{region '#Template'}
	{attribute 'Version' := '6.0.0.0'}
	{attribute 'Tags' := '"LCID": "1031", "Text": "AC, Plant, AHU, Lüftungsanlage"'}
	{attribute 'Tags' := '"LCID": "1033", "Text": "AC, Plant, AHU, Air handling unit"'}
	{attribute 'Using' := '"Type": "Template", "URI": "Priority"'}		 
	{attribute 'Using' := '"Type": "Template", "URI": "Site"'}
	{attribute 'Using' := '"Type": "Template", "URI": "E_BA_AC_OpMod01"'}
	{attribute 'Using' := '"Type": "Template", "URI": "E_BA_AC_PlantStep01"'}
	{attribute 'Description' := '"LCID": "1031", "Text": "Ventilator druckgesteuert, Einfache Abluft/Zuluftkaskade, Vorerhitzer, ERC Platte, Kühler "'}
	{attribute 'Description' := '"LCID": "1033", "Text": "Fan pressure controlled, Simple extract air/supply air cascade, PreHeater, ERC Plate, Cooler"'}
{endregion}
FUNCTION_BLOCK FB_BA_AHU_1st_10 EXTENDS FB_BA_View
VAR_INPUT CONSTANT	
	TOuA					: FB_BA_SensorAnalog;			
	TExhA					: FB_BA_SensorAnalog;	
	TSuA					: FB_BA_SensorAnalog;	
	TExtA					: FB_BA_SensorAnalog;								
	TRm						: FB_BA_SensorAnalog;	

	DiffPrssOuAFilt			: FB_BA_SensorAnalog;											
	FiltOuAMonit			: FB_BA_Hys_21;							
	DiffPrssExtAFilt		: FB_BA_SensorAnalog;				
	FiltExtAMonit			: FB_BA_Hys_21;	

	OuADmp					: FB_BA_AC_Dmp2P;	
	SuAPrss					: FB_BA_SensorAnalog;	
	SuADiffPrss				: FB_BA_SensorAnalog;		
	SuAFan					: FB_BA_AC_FanCtl;	
	SuADiffPrssMonit		: FB_BA_FdbAnalog;								

	ExhADmp					: FB_BA_AC_Dmp2P;	
	ExtAPrss				: FB_BA_SensorAnalog;	
	ExtADiffPrss			: FB_BA_SensorAnalog;		
	ExtAFan					: FB_BA_AC_FanCtl;								
	ExtADiffPrssMonit		: FB_BA_FdbAnalog;

	PreHtr					: FB_BA_AC_PreHtr;	
	Erc						: FB_BA_AC_ErcPl_02;								
	Col						: FB_BA_AC_ColT_02;								

	SpTRm					: FB_BA_Scale_04_Y2_3;	
	TCasCtrl				: FB_BA_AC_TCasCtrl_01;										 								

	SumNgtCol				: FB_BA_AC_SumNgtCol;	
	OpMod					: FB_BA_AC_OpMod1St;	

	PlantLock				: FB_BA_PlantLock;	

	PlantCmd				: FB_BA_AC_PlantCmd_AHU_1st_10;	

	TSeqLink				: FB_BA_AC_SeqT;
	stTSeqLink				: ST_BA_SeqLink;	//	Sequenz Link Struktur	//	Sequence link structure		
	
	arrAggregate			: ARRAY [1..MAX(1,BA_Param.nMaxAggregate)] OF ST_BA_Aggregate;

END_VAR
VAR // added by the converter: edge detectors and wires of the graphical bodies
    _w1 : ANY;
END_VAR

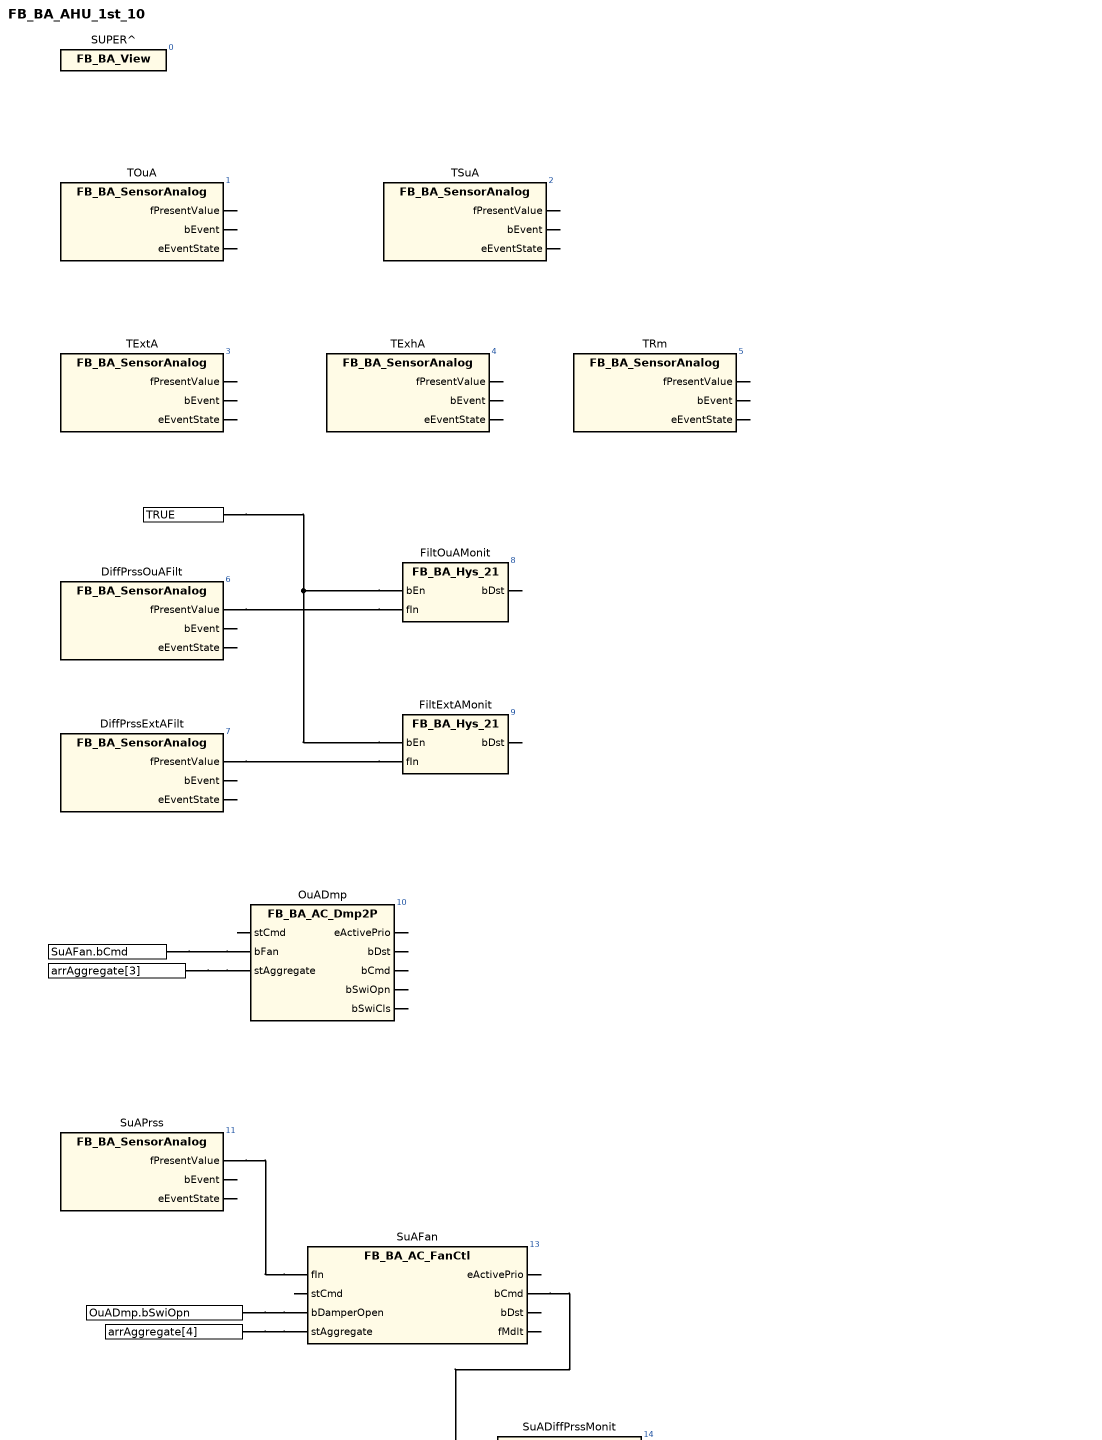
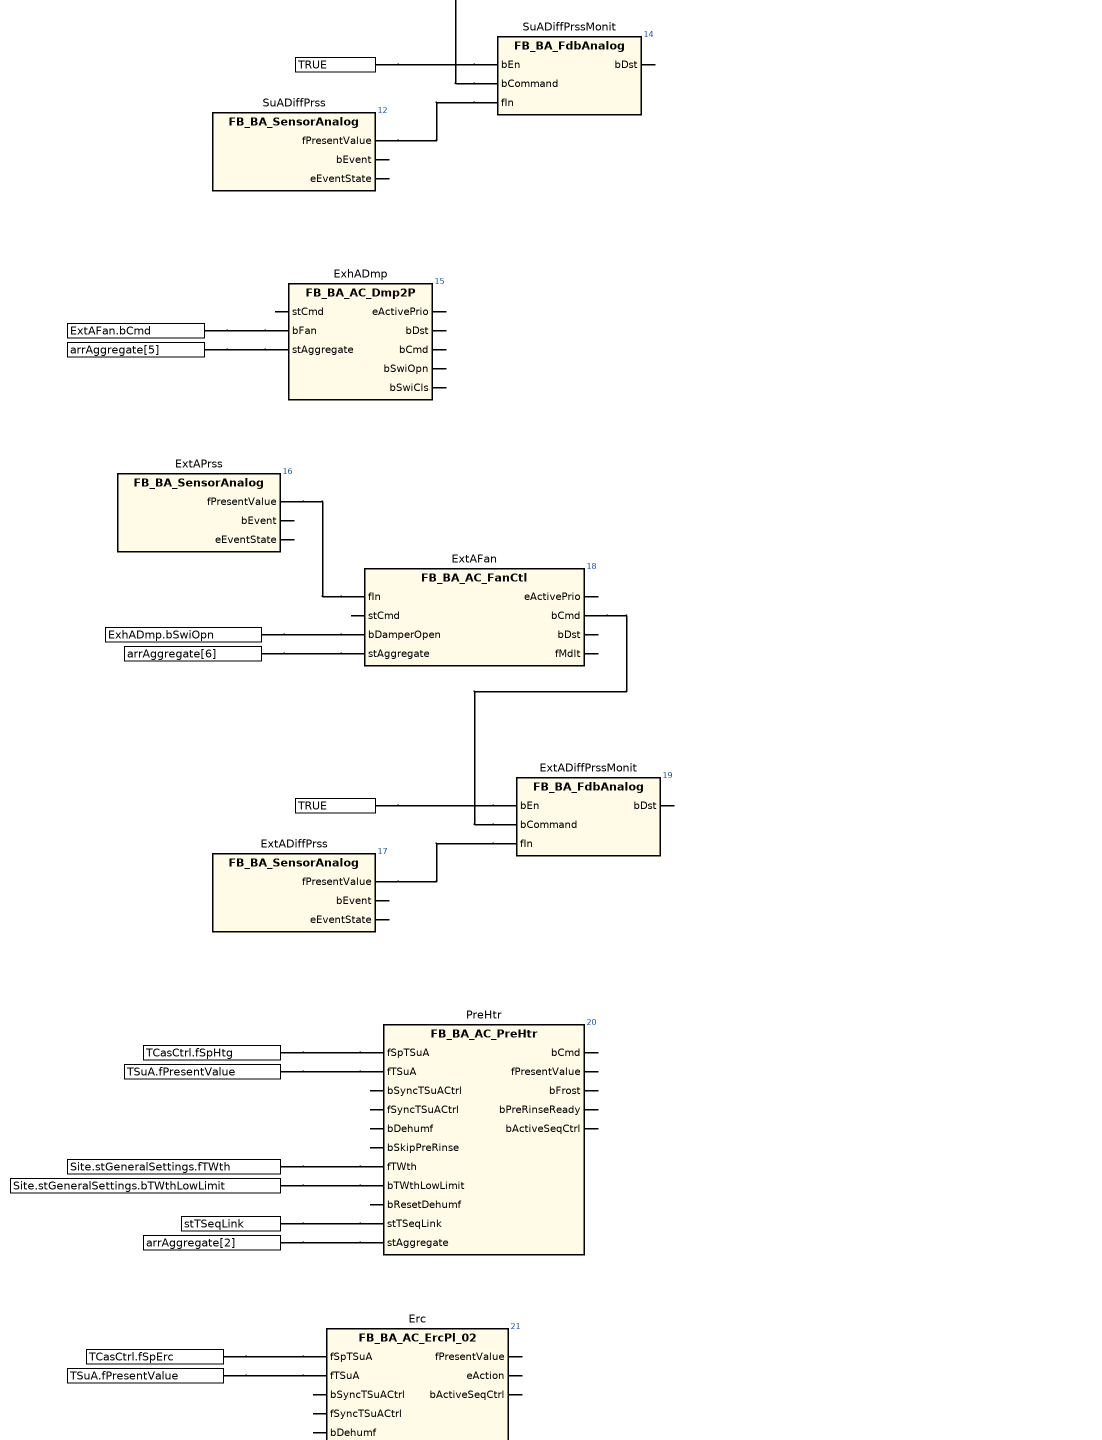
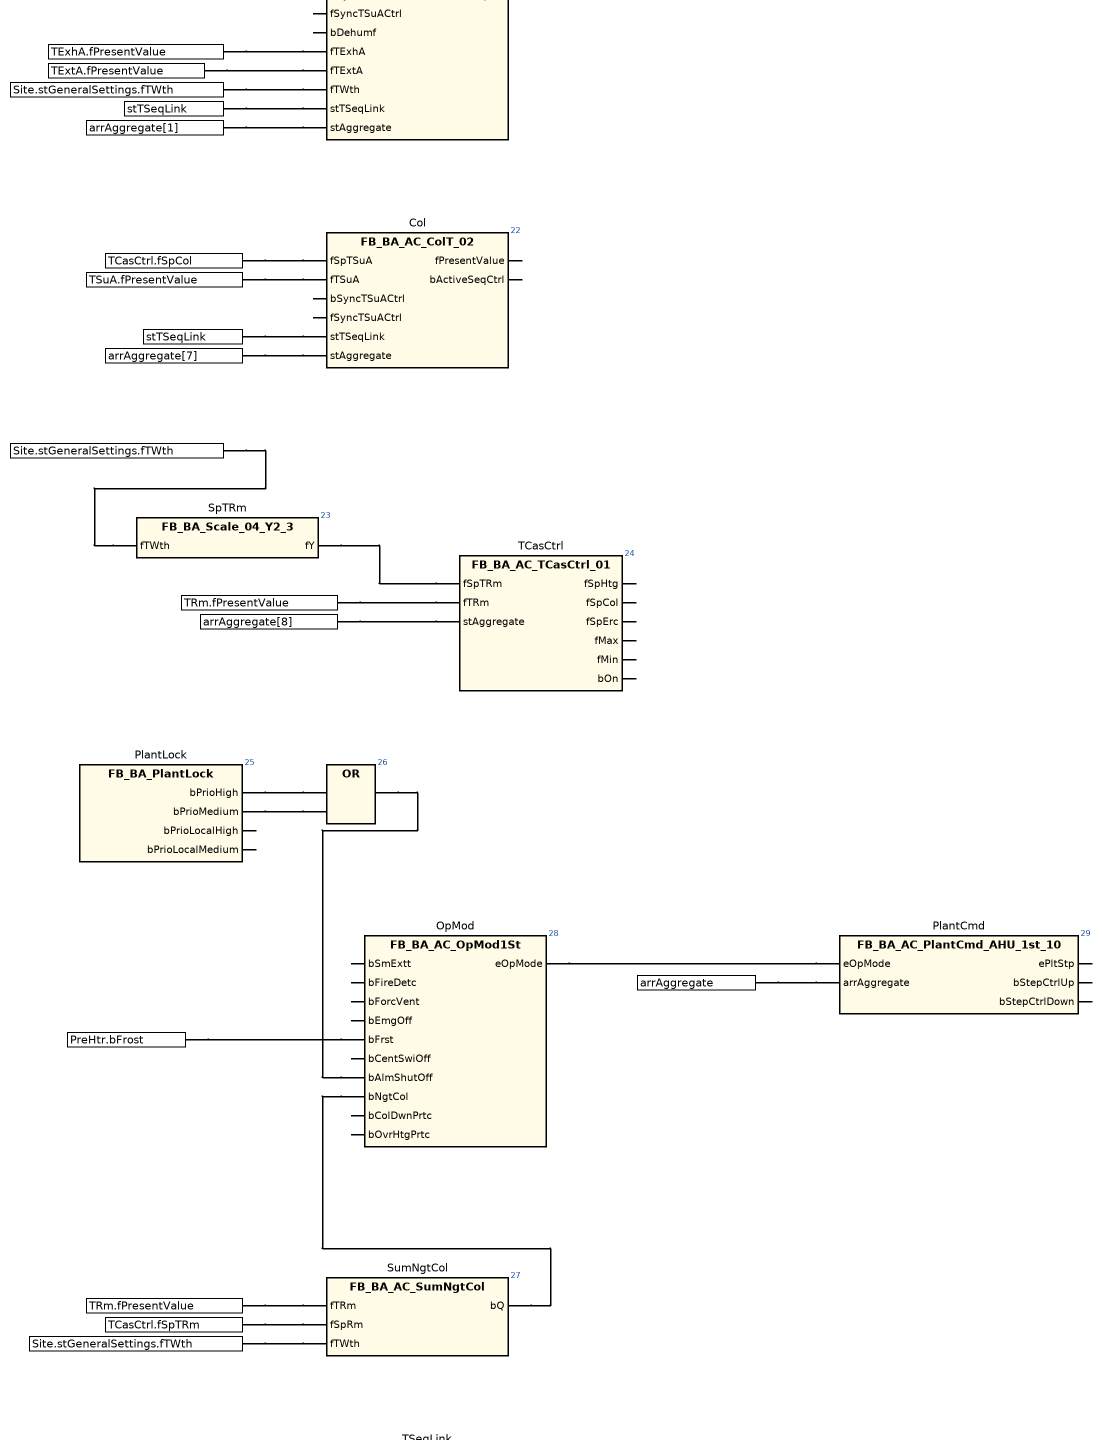
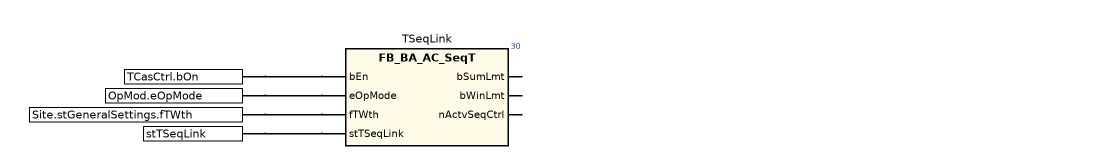
SUPER^(); // FB_BA_View
TOuA(); // FB_BA_SensorAnalog
TSuA(); // FB_BA_SensorAnalog
TExtA(); // FB_BA_SensorAnalog
TExhA(); // FB_BA_SensorAnalog
TRm(); // FB_BA_SensorAnalog
DiffPrssOuAFilt(); // FB_BA_SensorAnalog
DiffPrssExtAFilt(); // FB_BA_SensorAnalog
FiltOuAMonit(bEn := TRUE, fIn := DiffPrssOuAFilt.fPresentValue); // FB_BA_Hys_21
FiltExtAMonit(bEn := TRUE, fIn := DiffPrssExtAFilt.fPresentValue); // FB_BA_Hys_21
OuADmp(bFan := SuAFan.bCmd, stAggregate := arrAggregate[3]); // FB_BA_AC_Dmp2P
SuAPrss(); // FB_BA_SensorAnalog
SuADiffPrss(); // FB_BA_SensorAnalog
SuAFan(fIn := SuAPrss.fPresentValue, bDamperOpen := OuADmp.bSwiOpn, stAggregate := arrAggregate[4]); // FB_BA_AC_FanCtl
SuADiffPrssMonit(bEn := TRUE, bCommand := SuAFan.bCmd, fIn := SuADiffPrss.fPresentValue); // FB_BA_FdbAnalog
ExhADmp(bFan := ExtAFan.bCmd, stAggregate := arrAggregate[5]); // FB_BA_AC_Dmp2P
ExtAPrss(); // FB_BA_SensorAnalog
ExtADiffPrss(); // FB_BA_SensorAnalog
ExtAFan(fIn := ExtAPrss.fPresentValue, bDamperOpen := ExhADmp.bSwiOpn, stAggregate := arrAggregate[6]); // FB_BA_AC_FanCtl
ExtADiffPrssMonit(bEn := TRUE, bCommand := ExtAFan.bCmd, fIn := ExtADiffPrss.fPresentValue); // FB_BA_FdbAnalog
PreHtr(
    fSpTSuA := TCasCtrl.fSpHtg,
    fTSuA := TSuA.fPresentValue,
    fTWth := Site.stGeneralSettings.fTWth,
    bTWthLowLimit := Site.stGeneralSettings.bTWthLowLimit,
    stTSeqLink := stTSeqLink,
    stAggregate := arrAggregate[2]); // FB_BA_AC_PreHtr
Erc(
    fSpTSuA := TCasCtrl.fSpErc,
    fTSuA := TSuA.fPresentValue,
    fTExhA := TExhA.fPresentValue,
    fTExtA := TExtA.fPresentValue,
    fTWth := Site.stGeneralSettings.fTWth,
    stTSeqLink := stTSeqLink,
    stAggregate := arrAggregate[1]); // FB_BA_AC_ErcPl_02
Col(
    fSpTSuA := TCasCtrl.fSpCol,
    fTSuA := TSuA.fPresentValue,
    stTSeqLink := stTSeqLink,
    stAggregate := arrAggregate[7]); // FB_BA_AC_ColT_02
SpTRm(fTWth := Site.stGeneralSettings.fTWth); // FB_BA_Scale_04_Y2_3
TCasCtrl(fSpTRm := SpTRm.fY, fTRm := TRm.fPresentValue, stAggregate := arrAggregate[8]); // FB_BA_AC_TCasCtrl_01
PlantLock(); // FB_BA_PlantLock
_w1 := PlantLock.bPrioHigh OR PlantLock.bPrioMedium;
SumNgtCol(fTRm := TRm.fPresentValue, fSpRm := TCasCtrl.fSpTRm, fTWth := Site.stGeneralSettings.fTWth); // FB_BA_AC_SumNgtCol
OpMod(bFrst := PreHtr.bFrost, bAlmShutOff := _w1, bNgtCol := SumNgtCol.bQ); // FB_BA_AC_OpMod1St
PlantCmd(eOpMode := OpMod.eOpMode, arrAggregate := arrAggregate); // FB_BA_AC_PlantCmd_AHU_1st_10
TSeqLink(
    bEn := TCasCtrl.bOn,
    eOpMode := OpMod.eOpMode,
    fTWth := Site.stGeneralSettings.fTWth,
    stTSeqLink := stTSeqLink); // FB_BA_AC_SeqT

METHOD FB_init : BOOL
VAR_INPUT
	bInitRetains : BOOL; // if TRUE, the retain variables are initialized (warm start / cold start)
	bInCopyCode : BOOL;  // if TRUE, the instance afterwards gets moved into the copy code (online change)
END_VAR
PlantLock.Parent							:= THIS^;		

TOuA.iParent								:= THIS^;
TOuA.iLabel									:= LblAgg_TemperatureOutside; 		
TOuA.eDPADMode								:= E_BA_DPADMode.eInclude;										
TOuA.MV.eUnit								:= E_BA_Unit.eTemperature_DegreesCelsius;
TOuA.MV.fResolution 						:= 0.01;
TOuA.MV.fScaleOffset 						:= 0; 
TOuA.MV.bEventDetectionEnable				:= TRUE;
TOuA.MV.eEnPlantLock						:= E_BA_LockPriority.eNoLock;

TExhA.iParent								:= THIS^;		
TExhA.iLabel								:= LblAgg_TemperatureExhaustAir; 		
TExhA.eDPADMode								:= E_BA_DPADMode.eInclude;										
TExhA.MV.eUnit								:= E_BA_Unit.eTemperature_DegreesCelsius;
TExhA.MV.fResolution 						:= 0.01;
TExhA.MV.fScaleOffset 						:= 0; 
TExhA.MV.bEventDetectionEnable				:= TRUE;
TExhA.MV.eEnPlantLock						:= E_BA_LockPriority.eNoLock;

TSuA.iParent								:= THIS^;		
TSuA.iLabel									:= LblAgg_TemperatureSupplyAir; 	
TSuA.eDPADMode								:= E_BA_DPADMode.eInclude;										
TSuA.MV.eUnit								:= E_BA_Unit.eTemperature_DegreesCelsius;
TSuA.MV.fResolution 						:= 0.01;
TSuA.MV.fScaleOffset 						:= 0; 
TSuA.MV.bEventDetectionEnable				:= TRUE;
TSuA.MV.eEnPlantLock						:= E_BA_LockPriority.eMedium;

TExtA.iParent								:= THIS^;
TExtA.iLabel								:= LblAgg_TemperatureExtractAir; 	
TExtA.eDPADMode								:= E_BA_DPADMode.eInclude;										
TExtA.MV.eUnit								:= E_BA_Unit.eTemperature_DegreesCelsius;
TExtA.MV.fResolution 						:= 0.01;
TExtA.MV.fScaleOffset 						:= 0; 
TExtA.MV.bEventDetectionEnable				:= TRUE;
TExtA.MV.eEnPlantLock						:= E_BA_LockPriority.eNoLock;

TRm.iParent									:= THIS^;		
TRm.iLabel									:= LblAgg_TemperatureRoomAir; 	
TRm.eDPADMode								:= E_BA_DPADMode.eInclude;										
TRm.MV.eUnit								:= E_BA_Unit.eTemperature_DegreesCelsius;
TRm.MV.fResolution 							:= 0.01;
TRm.MV.fScaleOffset 						:= 0;
TRm.MV.bEventDetectionEnable				:= TRUE;
TRm.MV.eEnPlantLock							:= E_BA_LockPriority.eNoLock;

DiffPrssOuAFilt.iParent								:= THIS^;		 
DiffPrssOuAFilt.iLabel								:= LblAgg_PressureDifferentialOutsideAirFilter; 	
DiffPrssOuAFilt.sObjectName							:= '{Idx=03}';
DiffPrssOuAFilt.eDPADMode							:= E_BA_DPADMode.eInclude;										
DiffPrssOuAFilt.MV.eUnit							:= E_BA_Unit.ePressure_Pascals;
DiffPrssOuAFilt.MV.fResolution 						:= 0.03051851;
DiffPrssOuAFilt.MV.fScaleOffset 					:= 0; 
DiffPrssOuAFilt.MV.bEventDetectionEnable			:= TRUE;
DiffPrssOuAFilt.MV.eEnPlantLock						:= E_BA_LockPriority.eNoLock;

FiltOuAMonit.iParent								:= THIS^;
FiltOuAMonit.iLabel									:= LblAgg_AirFilterOutsideAir; 	
FiltOuAMonit.sObjectName							:= '{Idx=01}';
FiltOuAMonit.eDPADMode								:= E_BA_DPADMode.eInclude;
FiltOuAMonit.DstPreAlarm.bEventDetectionEnable		:= TRUE;
FiltOuAMonit.DstPreAlarm.eEnPlantLock				:= E_BA_LockPriority.eNoLock;	
FiltOuAMonit.DstMainAlarm.bEventDetectionEnable		:= TRUE;
FiltOuAMonit.DstMainAlarm.eEnPlantLock				:= E_BA_LockPriority.eMedium;

DiffPrssExtAFilt.iParent							:= THIS^;		
DiffPrssExtAFilt.iLabel								:= LblAgg_PressureDifferentialExtractAirFilter; 	
DiffPrssExtAFilt.sObjectName						:= '{Idx=04}';
DiffPrssExtAFilt.eDPADMode							:= E_BA_DPADMode.eInclude;										
DiffPrssExtAFilt.MV.eUnit							:= E_BA_Unit.ePressure_Pascals;
DiffPrssExtAFilt.MV.fResolution 					:= 0.03051851;
DiffPrssExtAFilt.MV.fScaleOffset 					:= 0; 
DiffPrssExtAFilt.MV.bEventDetectionEnable			:= TRUE;
DiffPrssExtAFilt.MV.eEnPlantLock					:= E_BA_LockPriority.eNoLock;

FiltExtAMonit.iParent								:= THIS^;
FiltExtAMonit.iLabel								:= LblAgg_AirFilterExtractAir; 		
FiltExtAMonit.sObjectName							:= '{Idx=02}';						 
FiltExtAMonit.eDPADMode								:= E_BA_DPADMode.eInclude;
FiltExtAMonit.DstPreAlarm.bEventDetectionEnable		:= TRUE;
FiltExtAMonit.DstPreAlarm.eEnPlantLock				:= E_BA_LockPriority.eNoLock;	
FiltExtAMonit.DstMainAlarm.bEventDetectionEnable	:= TRUE;
FiltExtAMonit.DstMainAlarm.eEnPlantLock				:= E_BA_LockPriority.eMedium;			

OuADmp.iParent								:= THIS^;
OuADmp.iLabel								:= LblAgg_VentilationDamperOutsideAir; 
OuADmp.sObjectName							:= '{Idx=01}';						 
OuADmp.eDPADMode							:= E_BA_DPADMode.eInclude;
OuADmp.MonitOpen.Dst.eEnPlantLock			:= E_BA_LockPriority.eMedium;
OuADmp.MonitOpen.Dst.bEventDetectionEnable	:= TRUE;						
OuADmp.MonitClose.Dst.eEnPlantLock			:= E_BA_LockPriority.eNoLock;								
OuADmp.MonitClose.Dst.bEventDetectionEnable	:= TRUE;						

SuAPrss.iParent								:= THIS^;
SuAPrss.iLabel								:= LblAgg_PressureSupplyAir; 
SuAPrss.sObjectName							:= '{Idx=01}';						 
SuAPrss.eDPADMode							:= E_BA_DPADMode.eInclude;																						
SuAPrss.MV.eUnit							:= E_BA_Unit.ePressure_Pascals;
SuAPrss.MV.fResolution 						:= 0.03051851;
SuAPrss.MV.fScaleOffset 					:= 0;
SuAPrss.MV.bEventDetectionEnable			:= TRUE;
SuAPrss.MV.eEnPlantLock						:= E_BA_LockPriority.eNoLock;

SuADiffPrss.iParent							:= THIS^;		
SuADiffPrss.iLabel							:= LblAgg_PressureDifferentialSupplyAirFan; 
SuADiffPrss.sObjectName						:= '{Idx=01}';						 
SuADiffPrss.eDPADMode						:= E_BA_DPADMode.eInclude;																						
SuADiffPrss.MV.eUnit						:= E_BA_Unit.ePressure_Pascals;
SuADiffPrss.MV.fResolution 					:= 0.03051851;
SuADiffPrss.MV.fScaleOffset 				:= 0; 
SuADiffPrss.MV.bEventDetectionEnable		:= TRUE;
SuADiffPrss.MV.eEnPlantLock					:= E_BA_LockPriority.eNoLock;

SuAFan.iParent								:= THIS^;
SuAFan.iLabel								:= LblAgg_FanSupplyAir; 								 
SuAFan.sObjectName							:= '{Idx=01}';						 
SuAFan.eDPADMode							:= E_BA_DPADMode.eInclude;								
SuAFan.Dst.eEnPlantLock						:= E_BA_LockPriority.eMedium;
SuAFan.Dst.bEventDetectionEnable			:= TRUE;
SuAFan.ThOvrld.eEnPlantLock					:= E_BA_LockPriority.eMedium;	
SuAFan.ThOvrld.bEventDetectionEnable		:= TRUE;
SuAFan.MntnSwi.eEnPlantLock					:= E_BA_LockPriority.eMedium;
SuAFan.MntnSwi.bEventDetectionEnable		:= TRUE;

SuADiffPrssMonit.iParent					:= THIS^;
SuADiffPrssMonit.iLabel						:= LblCtl_DifferencePressureMonitoringSupplyAirFan; 												 
SuADiffPrssMonit.sObjectName				:= '{Idx=01}';						 
SuADiffPrssMonit.eDPADMode					:= E_BA_DPADMode.eInclude;
SuADiffPrssMonit.Dst.bEventDetectionEnable	:= TRUE;								
SuADiffPrssMonit.Dst.eEnPlantLock			:= E_BA_LockPriority.eMedium;				

ExhADmp.iParent								:= THIS^;
ExhADmp.iLabel								:= LblAgg_VentilationDamperExhaustAir; 							 
ExhADmp.sObjectName							:= '{Idx=02}';						 
ExhADmp.eDPADMode							:= E_BA_DPADMode.eInclude;								
ExhADmp.MonitOpen.Dst.eEnPlantLock			:= E_BA_LockPriority.eMedium;								
ExhADmp.MonitOpen.Dst.bEventDetectionEnable	:= TRUE;						
ExhADmp.MonitClose.Dst.eEnPlantLock			:= E_BA_LockPriority.eNoLock;				
ExhADmp.MonitClose.Dst.bEventDetectionEnable:= TRUE;	

ExtAPrss.iParent							:= THIS^;
ExtAPrss.iLabel								:= LblAgg_PressureExtractAir; 						
ExtAPrss.sObjectName						:= '{Idx=01}';						 
ExtAPrss.eDPADMode							:= E_BA_DPADMode.eInclude;																						
ExtAPrss.MV.eUnit							:= E_BA_Unit.ePressure_Pascals;
ExtAPrss.MV.fResolution 					:= 0.03051851;
ExtAPrss.MV.fScaleOffset 					:= 0; 
ExtAPrss.MV.bEventDetectionEnable			:= TRUE;
ExtAPrss.MV.eEnPlantLock					:= E_BA_LockPriority.eNoLock;

ExtADiffPrss.iParent						:= THIS^;
ExtADiffPrss.iLabel							:= LblAgg_PressureDifferentialExtractAirFan; 
ExtADiffPrss.sObjectName					:= '{Idx=02}';						 
ExtADiffPrss.eDPADMode						:= E_BA_DPADMode.eInclude;																						
ExtADiffPrss.MV.eUnit						:= E_BA_Unit.ePressure_Pascals;
ExtADiffPrss.MV.fResolution 				:= 0.03051851;
ExtADiffPrss.MV.fScaleOffset 				:= 0; 
ExtADiffPrss.MV.bEventDetectionEnable		:= TRUE;
ExtADiffPrss.MV.eEnPlantLock				:= E_BA_LockPriority.eNoLock;

ExtAFan.iParent								:= THIS^;
ExtAFan.iLabel								:= LblAgg_FanExtractAir; 
ExtAFan.sObjectName							:= '{Idx=01}';						 
ExtAFan.eDPADMode							:= E_BA_DPADMode.eInclude;								
ExtAFan.Dst.eEnPlantLock					:= E_BA_LockPriority.eMedium;
ExtAFan.Dst.bEventDetectionEnable			:= TRUE;
ExtAFan.ThOvrld.eEnPlantLock				:= E_BA_LockPriority.eMedium;	
ExtAFan.ThOvrld.bEventDetectionEnable		:= TRUE;
ExtAFan.MntnSwi.eEnPlantLock				:= E_BA_LockPriority.eMedium;
ExtAFan.MntnSwi.bEventDetectionEnable		:= TRUE;

ExtADiffPrssMonit.iParent					:= THIS^; 
ExtADiffPrssMonit.iLabel					:= LblCtl_DifferencePressureMonitoringExtractAirFan; 
ExtADiffPrssMonit.sObjectName				:= '{Idx=02}';						 
ExtADiffPrssMonit.eDPADMode					:= E_BA_DPADMode.eInclude;								
ExtADiffPrssMonit.Dst.bEventDetectionEnable	:= TRUE;										
ExtADiffPrssMonit.Dst.eEnPlantLock			:= E_BA_LockPriority.eMedium;													

SpTRm.iParent								:= THIS^;
SpTRm.iLabel								:= LblCtl_TSetpointCalculation; 	
SpTRm.sObjectName							:= '{Idx=01}';						 						 
SpTRm.eDPADMode								:= E_BA_DPADMode.eInclude;								

TCasCtrl.iParent							:= THIS^;
TCasCtrl.iLabel								:= LblCtl_TCascadeSupplyAirControl; 
TCasCtrl.sObjectName						:= '{Idx=01}';						 
TCasCtrl.eDPADMode							:= E_BA_DPADMode.eInclude;																		 								

SumNgtCol.iParent							:= THIS^; 
SumNgtCol.iLabel							:= LblCtl_SummerNightCooling; 	
SumNgtCol.sObjectName						:= '{Idx=01}';						 
SumNgtCol.eDPADMode							:= E_BA_DPADMode.eInclude;								

OpMod.iParent								:= THIS^;
OpMod.iLabel								:= LblCtl_OperationMode; 
OpMod.sObjectName							:= '{Idx=01}';						 
OpMod.eDPADMode								:= E_BA_DPADMode.eInclude;		

PreHtr.iParent										:= THIS^;
PreHtr.iLabel										:= LblCtl_PreHeater; 
PreHtr.sObjectName									:= '{Idx=01}';						 
PreHtr.eDPADMode									:= E_BA_DPADMode.eIncludeDescription;								
PreHtr.TFl.MV.bEventDetectionEnable					:= TRUE;
PreHtr.TRt.MV.eEnPlantLock							:= E_BA_LockPriority.eMedium;
PreHtr.TRt.MV.bEventDetectionEnable					:= TRUE;
PreHtr.TRtCtrl.PreRinseDst.eEnPlantLock				:= E_BA_LockPriority.eNoLock;
PreHtr.TRtCtrl.PreRinseDst.bEventDetectionEnable	:= TRUE;
PreHtr.TFrost.MV.eEnPlantLock						:= E_BA_LockPriority.eMedium;
PreHtr.TFrost.MV.bEventDetectionEnable				:= TRUE;
PreHtr.FrostThermostat.Input.eEnPlantLock			:= E_BA_LockPriority.eMedium;	
PreHtr.FrostThermostat.Input.bEventDetectionEnable	:= TRUE;	
PreHtr.Pu.Dst.eEnPlantLock							:= E_BA_LockPriority.eMedium;
PreHtr.Pu.Dst.bEventDetectionEnable					:= TRUE;

Erc.iParent									:= THIS^; 
Erc.iLabel									:= LblCtl_EnergyRecovery; 
Erc.sObjectName								:= '{Idx=01}';						 
Erc.eDPADMode								:= E_BA_DPADMode.eIncludeDescription;																
Erc.DiffPrssSwi.Input.bEventDetectionEnable	:= TRUE;

Col.iParent									:= THIS^;
Col.iLabel									:= LblCtl_Cooler; 
Col.sObjectName								:= '{Idx=01}';						 
Col.eDPADMode								:= E_BA_DPADMode.eIncludeDescription;								
Col.TFl.MV.bEventDetectionEnable			:= TRUE;
Col.TRt.MV.bEventDetectionEnable			:= TRUE;			

PlantCmd.iParent							:= THIS^;
PlantCmd.iLabel								:= LblCtl_PlantStartUp;
PlantCmd.sObjectName						:= '{Idx=01}';						 
PlantCmd.eDPADMode							:= E_BA_DPADMode.eInclude;			

TSeqLink.iParent							:= THIS^;
TSeqLink.iLabel								:= LblCtl_TSequenceControl;   
TSeqLink.sObjectName						:= '{Idx=01}';						 
TSeqLink.eDPADMode							:= E_BA_DPADMode.eInclude;
END_METHOD

END_FUNCTION_BLOCK

(* stored: Version 1.1.0.1, ProductVersion 3.1.4024.12
   POU FB_BA_AHU_1st_10: Id {d65262ba-4bba-44a3-a324-7b56b64582b9}, SpecialFunc None
   Method FB_init: Id {117b0697-8883-45fa-9f9c-d79a25fd0d56} *)
